PROGRAM POU_Master_Calib_2
VAR
	criteria: REAL := 0.5; // Acceptance Criteria (0.1 ~ 5.0)
	failures: INT := 0; // Allowable Failures (0 ~ 5)
	targetVolume: REAL := 0.50; // Volume Target (mL)
	replicates: INT := 5; // Number of checks (0 ~ 10)
	tareWt: REAL; //Weight before
	grossWt: REAL; //Weight after
	netWt: REAL; // rsult of (grossWt - tareWt)
	netVolume: REAL; //result of (netWt * density)
	state: INT;
	valveNo: INT;
	pumpNo: INT:=1;
	timeWt: ton;
	timer2: ton;
	timer3: ton;
	selectPump: ARRAY[1..10] OF STRING;
	result: ARRAY[1..10] OF ST_Results;
	start: BOOL;
	stop: BOOL;
	movimentDONE: BOOL;
	revs: REAL;
	valvePos: USINT;
	repli: INT:= 1;
	axiPower: MC_Power;
	i: INT;
	scale: FB_ScaleDevice;
	adjust: ARRAY[1..10] OF BOOL;
	correctRev: REAL;
	enableAdj: BOOL;
	opening: REAL;
	runLinear: BOOL;
	adjustSum: REAL;
	recResult: int:=1;
END_VAR

timeWt();
timer2();
timer3();

IF stop THEN
	powerOFF();
	stop:=FALSE;
END_IF

IF pumpNo = 1 OR pumpNo = 2 THEN
	valveNo:= 1;
ELSIF pumpNo = 3 OR pumpNo = 4 THEN
	valveNo:= 2;
ELSIF pumpNo = 5 OR pumpNo = 6 THEN
	valveNo:= 3;
ELSIF pumpNo = 7 OR pumpNo = 8 THEN
	valveNo:= 4;
ELSIF pumpNo = 9 OR pumpNo = 10 THEN
	valveNo:= 5;
END_IF

CASE state OF
	
0: //Idle
	IF start THEN
		GVL_Marco.revs:= GVL_Marco.mL_target;
		GVL_Marco.valvPos:= 6;
		timeWt(in:=TRUE, pt:=T#10S);
		repli:= 1;
		recResult:= 1;
		
		FOR i:= 1 TO 10 BY 1 DO
			GVL_Marco.resetAxi[i]:= FALSE;
			GVL_Marco.enableAxi[i]:= TRUE;
		END_FOR 
		
		FOR i:= 1 TO 5 BY 1 DO
			GVL_Marco.enableValv[i]:= TRUE;		
		END_FOR
		
		FOR i:=1 TO 50 BY 1 DO
			GVL_Marco.calibResult[i].grossWt:=0;
			GVL_Marco.calibResult[i].netWt:=0;
			GVL_Marco.calibResult[i].pumpNo:=0;
			GVL_Marco.calibResult[i].tareWt:=0;
		END_FOR
		
		state:= 10;
	ELSE
		state:= 0;
	END_IF
	
10:	//Enable the pump motor
	
	IF GVL_Motion.aValves[1].Axis.Status.InTargetPosition AND
		GVL_Motion.aValves[2].Axis.Status.InTargetPosition AND
		GVL_Motion.aValves[3].Axis.Status.InTargetPosition AND
		GVL_Motion.aValves[4].Axis.Status.InTargetPosition AND
		GVL_Motion.aValves[5].Axis.Status.InTargetPosition AND timeWt.Q THEN
		FOR i:= 1 TO 5 BY 1 DO
			GVL_Marco.enableValv[i]:= FALSE;		
		END_FOR
		timeWt(in:=FALSE);
		state:= 20;
	ELSE
		state:= 10;
	END_IF		

20:	//Fill the Jars from Box
	
	IF NOT GVL_Motion.aPumps[pumpNo].Rotary.Axis.Status.Disabled THEN
		
		revs:= GVL_Marco.revs*2;
		GVL_Marco.runFWD[pumpNo]:= TRUE;
		
		start:= FALSE;
		timer2(in:=TRUE, pt:=T#10S);
		state:= 30;
	ELSE
		state:= 20;
	END_IF

30: //Move valve to position 6
	
	IF NOT GVL_Motion.aPumps[pumpNo].Rotary.Axis.Status.Moving AND timer2.Q THEN
		
		GVL_Marco.valvPos:= 6;
		timer2(in:=FALSE);
		timeWt(in:=TRUE, pt:=T#10S);
		
		GVL_Marco.runFWD[pumpNo]:= FALSE;
		
		FOR i:=1 TO 5 BY 1 DO
			GVL_Marco.enableValv[i]:= TRUE;
		END_FOR
		
		
		state:= 40;
		
	ELSE
		state:= 30;
	END_IF


40: //Fill the calibration box(setup) - NO MORE

	IF GVL_Motion.aValves[1].Axis.Status.InTargetPosition AND
		GVL_Motion.aValves[2].Axis.Status.InTargetPosition AND
		GVL_Motion.aValves[3].Axis.Status.InTargetPosition AND
		GVL_Motion.aValves[4].Axis.Status.InTargetPosition AND
		GVL_Motion.aValves[5].Axis.Status.InTargetPosition AND timeWt.Q THEN
		
		FOR i:= 1 TO 5 BY 1 DO
			GVL_Marco.enableValv[i]:= FALSE;
		END_FOR
		
		//revs:= GVL_Marco.revs/2;
		//GVL_Marco.runBWD[pumpNo]:= TRUE;
		
		timeWt(in:=FALSE);
		timer2(in:=TRUE, pt:=T#10S);
		state:= 50;
		
	ELSE
		state:= 40;	
	END_IF

50: //Waiting

	IF NOT GVL_Motion.aPumps[pumpNo].Rotary.Axis.Status.Moving AND timer2.Q THEN
		GVL_Marco.runBWD[pumpNo]:= FALSE;
		timer2(in:=FALSE);
		timeWt(in:=TRUE, pt:=T#10S);
		GVL_Calibration.fbScaleDevice.RequestWeight();
		state:= 55;
	ELSE
		state:= 50;
	END_IF
	
55: //Make Tara
	
	IF timeWt.Q THEN
		tareWt:= GVL_Calibration.fbScaleDevice.RequestWeight();
		timeWt(in:=FALSE);
		state:= 60;
	ELSE
		state:= 55;
	END_IF
	
60: //Fill box from jar

	IF tareWt <> 9999.0 THEN
		GVL_Marco.calibResult[recResult].tareWt:= tareWt;
		revs:= GVL_Marco.revs;
		GVL_Marco.runBWD[pumpNo]:= TRUE;
		timer2(in:=TRUE, pt:=T#10S);
		state:= 70;
	ELSE
		state:= 60;
	END_IF
	
70: //Waiting

	IF NOT GVL_Motion.aPumps[pumpNo].Rotary.Axis.Status.Moving AND timer2.Q THEN
		GVL_Marco.runBWD[pumpNo]:= FALSE;
		timer2(in:=FALSE);
		timeWt(in:=TRUE, pt:=T#10S);
		GVL_Calibration.fbScaleDevice.RequestWeight();
		state:= 75;
	ELSE
		state:= 70;
	END_IF

75: //Get gross weight
	
	IF timeWt.Q THEN
		grossWt:= GVL_Calibration.fbScaleDevice.RequestWeight();
		timeWt(in:=FALSE);
		state:= 80;
	ELSE
		state:= 75;
	END_IF
	
80: //Return jar to box

	IF grossWt <> 9999.0 THEN
		GVL_Marco.calibResult[recResult].grossWt:= grossWt;
		GVL_Marco.calibResult[recResult].netWt:= GVL_Marco.calibResult[recResult].grossWt - GVL_Marco.calibResult[recResult].tareWt;
		GVL_Marco.calibResult[recResult].pumpNo:= pumpNo;
		recResult:= recResult +1;
			
		revs:= GVL_Marco.revs;
		GVL_Marco.runBWD[pumpNo]:= TRUE;

		timer3(in:=TRUE, pt:=T#10S);
		repli := repli +1; 
		state:= 90;
	ELSE
		state:= 80;
	END_IF

90: //Check replicates

	IF repli < replicates+1 AND timer3.Q AND GVL_Motion.aPumps[pumpNo].Rotary.Axis.Status.NotMoving THEN
		timer3(in:=FALSE);
		GVL_Marco.runBWD[pumpNo]:= FALSE;
		timer2(in:=TRUE, pt:=T#10S);
		state:= 50;
	ELSIF repli >= replicates AND timer3.Q AND GVL_Motion.aPumps[pumpNo].Rotary.Axis.Status.NotMoving THEN
		timer3(in:=FALSE);
		GVL_Marco.runBWD[pumpNo]:= FALSE;
		timer2(in:=TRUE, pt:=T#10S);
		state:= 100;
	ELSE
		state:= 90;
	END_IF

100: //Empty the jar to box

	IF  GVL_Motion.aValves[1].Axis.Status.InTargetPosition AND 
		GVL_Motion.aValves[2].Axis.Status.InTargetPosition AND
		GVL_Motion.aValves[3].Axis.Status.InTargetPosition AND
		GVL_Motion.aValves[4].Axis.Status.InTargetPosition AND
		GVL_Motion.aValves[5].Axis.Status.InTargetPosition AND timer2.Q THEN
		
		revs:= GVL_Marco.revs;
		IF pumpNo = 10 THEN
			GVL_Marco.runBWD[pumpNo]:= TRUE;
			state:= 110;
		ELSE
			pumpNo:= pumpNo + 1;
			repli:= 1;
			timer2(in:=TRUE, pt:=T#10S);
			state:= 20;
		END_IF
				
		timer2(in:=FALSE);
		timer3(in:=TRUE, pt:=T#10S);
		
	ELSE
		state:= 100;
	END_IF
	
110: //Done

	IF GVL_Motion.aPumps[1].Rotary.Axis.Status.NotMoving AND
		GVL_Motion.aPumps[2].Rotary.Axis.Status.NotMoving AND
		GVL_Motion.aPumps[3].Rotary.Axis.Status.NotMoving AND
		GVL_Motion.aPumps[4].Rotary.Axis.Status.NotMoving AND
		GVL_Motion.aPumps[5].Rotary.Axis.Status.NotMoving AND
		GVL_Motion.aPumps[6].Rotary.Axis.Status.NotMoving AND
		GVL_Motion.aPumps[7].Rotary.Axis.Status.NotMoving AND
		GVL_Motion.aPumps[8].Rotary.Axis.Status.NotMoving AND
		GVL_Motion.aPumps[9].Rotary.Axis.Status.NotMoving AND
		GVL_Motion.aPumps[10].Rotary.Axis.Status.NotMoving AND timer3.Q THEN
		FOR i:=1 TO 10 BY 1 DO
			GVL_Marco.runBWD[i]:= FALSE;
		END_FOR
		
		timer3(in:=FALSE);
		timeWt(in:=TRUE, pt:=T#10S);
		state:= 120;
	ELSE
		state:= 110;
	END_IF
	
120:

	IF GVL_Motion.aPumps[1].Rotary.Axis.Status.NotMoving AND
		GVL_Motion.aPumps[2].Rotary.Axis.Status.NotMoving AND
		GVL_Motion.aPumps[3].Rotary.Axis.Status.NotMoving AND
		GVL_Motion.aPumps[4].Rotary.Axis.Status.NotMoving AND
		GVL_Motion.aPumps[5].Rotary.Axis.Status.NotMoving AND
		GVL_Motion.aPumps[6].Rotary.Axis.Status.NotMoving AND
		GVL_Motion.aPumps[7].Rotary.Axis.Status.NotMoving AND
		GVL_Motion.aPumps[8].Rotary.Axis.Status.NotMoving AND
		GVL_Motion.aPumps[9].Rotary.Axis.Status.NotMoving AND
		GVL_Motion.aPumps[10].Rotary.Axis.Status.NotMoving AND timeWt.Q THEN
		FOR i:=1 TO 10 BY 1 DO
			GVL_Marco.resetAxi[i]:= TRUE;
			GVL_Marco.enableAxi[i]:= FALSE;
		END_FOR
		
		(*IF GVL_Marco.revs > GVL_Marco.mL_target THEN
			correctRev:= GVL_Marco.revs - GVL_Marco.mL_target;
		ELSIF GVL_Marco.revs < GVL_Marco.mL_target THEN
			correctRev:= GVL_Marco.mL_target - GVL_Marco.revs; 	
		END_IF*)
		state:= 0;
	ELSE
		state:= 120;
	END_IF
	
END_CASE

METHOD moveValve : BOOL
VAR
	state: INT;
	valveNo: INT;
END_VAR
VAR_INPUT
	pumNo: INT;
	valvePos: USINT;
	
END_VAR
IF pumpNo = 1 OR pumpNo = 2 THEN
	valveNo:= 1;
ELSIF pumpNo = 3 OR pumpNo = 4 THEN
	valveNo:= 2;
ELSIF pumpNo = 5 OR pumpNo = 6 THEN
	valveNo:= 3;
ELSIF pumpNo = 7 OR pumpNo = 8 THEN
	valveNo:= 4;
ELSIF pumpNo = 9 OR pumpNo = 10 THEN
	valveNo:= 5;
END_IF

GVL_Motion.aValvesObj[valveNo].MoveValve(iPosition := valvePos, rVelocity := GVL_Motion.aValves[1].rTargetVel, rAcc := GVL_Motion.aValves[1].rAcceleration, rDec := GVL_Motion.aValves[1].rDeceleration);

CASE state OF
	
0:

	IF NOT GVL_Motion.aValves[valveNo].Axis.Status.Moving THEN
		GVL_Motion.aValvesObj[valveNo].MoveValve(iPosition := valvePos, rVelocity := GVL_Motion.aValves[1].rTargetVel, rAcc := GVL_Motion.aValves[1].rAcceleration, rDec := GVL_Motion.aValves[1].rDeceleration);
		movimentDONE:=FALSE;
		state:= 1;
	ELSE
		state:= 0;	
	END_IF

1:
	IF NOT GVL_Motion.aValves[valveNo].Axis.Status.Moving THEN
			movimentDONE:= TRUE;
			State:= 0;
		ELSE
			state:= 1;
		END_IF
	
	
END_CASE
END_METHOD

METHOD powerOFF : BOOL
VAR
	axiPower: MC_Power;
	pumpNo: INT;
	
END_VAR
VAR_INPUT
	
	
END_VAR
FOR pumpNo:=1 TO 10 BY 1 DO
	axiPower(
	Axis:= GVL_Motion.aPumps[pumpNo].Rotary.Axis,
	Enable:= FALSE,
	Enable_Negative:= FALSE,
	Enable_Positive:= FALSE,
	Override:= 100);
	
	axiPower(
	Axis:= GVL_Motion.aPumps[pumpNo].Linear.Axis,
	Enable:= FALSE,
	Enable_Negative:= FALSE,
	Enable_Positive:= FALSE,
	Override:= 100);
END_FOR
END_METHOD

METHOD runBwd : BOOL
VAR
	moveRel: MC_MoveRelative;
	selectPosRel: LREAL;
	
END_VAR
VAR_INPUT
	pumpNo: INT;
	revs: INT;
	 
END_VAR

selectPosRel:= revs*360;

moveRel(
	Axis:= GVL_Motion.aPumps[pumpNo].Rotary.Axis,
	Execute:= TRUE,
	Distance:= selectPosRel*-1,
	Velocity:= 3000,
	Acceleration:= 3000,
	Deceleration:= 3000);
END_METHOD

METHOD runFwd : BOOL
VAR
	moveRel: MC_MoveRelative;
	selectPosRel: LREAL;
	
END_VAR
VAR_INPUT
	pumpNo: INT;
	revs: INT;
	 
END_VAR

selectPosRel:= revs*360;

moveRel(
	Axis:= GVL_Motion.aPumps[pumpNo].Rotary.Axis,
	Execute:= TRUE,
	Distance:= selectPosRel,
	Velocity:= 3000,
	Acceleration:= 3000,
	Deceleration:= 3000);
END_METHOD

END_PROGRAM

(* stored: Version 1.1.0.1, ProductVersion 3.1.4024.15
   POU POU_Master_Calib_2: Id {6bbea130-751c-482b-ab38-2633c1a032a0}, SpecialFunc None
   Method moveValve: Id {7d8274b1-957b-4011-8ef2-829aa21b82cd}
   Method powerOFF: Id {30b0883a-4a1b-467e-8465-76f56bd75b4b}
   Method runBwd: Id {eefadefd-fea3-4ebd-9d79-902f701041c8}
   Method runFwd: Id {1d946b5b-94f3-420d-aaf7-a77846e90b00} *)
